// TwinCAT 3 PLC project Untitled1
// ProgramVersion: 3.1.4024.0
// libraries:
//   Tc2_Standard, * (Beckhoff Automation GmbH)
//   Tc2_System, * (Beckhoff Automation GmbH)
//   Tc3_Module, * (Beckhoff Automation GmbH)
// project tree:
//   GVLs/ GVL.TcGVL
//   / PlcTask.TcTTO
//   POUs/ MAIN.TcPOU, PLC_FB.TcPOU
// real-time tasks:
//   TASK PlcTask: cycle T#1ms, priority 20, ADS port 350
// I/O:
//   DEVICE Device 1 (EtherCAT), AmsNetId 5.136.192.215.2.1
//     Term 1 (EK1200) [EK1200-5000 EtherCAT Power supply (2A E-Bus)]
//       Term 2 (EL3104) [EL3104 4Ch. Ana. Input +/-10V Diff.]
//       Term 3 (EL1018) [EL1018 8Ch. Dig. Input 24V, 10µs]
//       Term 4 (EL2008) [EL2008 8Ch. Dig. Output 24V, 0.5A]
//       Term 5 (EL2008) [EL2008 8Ch. Dig. Output 24V, 0.5A]
//       Term 6 (EL2008) [EL2008 8Ch. Dig. Output 24V, 0.5A]
//       Term 7 (EL3632) [EL3632 2Ch. IEPE Sensor]
//       Term 8 (EL3632) [EL3632 2Ch. IEPE Sensor]
//       Term 9 (EL9011) [EL9011 End Terminal]
//   DEVICE Device 4 (COM Port)
//   DEVICE Device 5 (NOV-DP-RAM)
// variable links:
//   Untitled1/Untitled1 Instance <-> Device 1 (EtherCAT)/Term 1 (EK1200)/Term 2 (EL3104)
//     PlcTask Inputs/GVL.GvlDataAll[31] <-> AI Standard Channel 1/Value
//     PlcTask Inputs/GVL.GvlDataAll[32] <-> AI Standard Channel 2/Value
//     PlcTask Inputs/GVL.GvlDataAll[33] <-> AI Standard Channel 3/Value
//   Untitled1/Untitled1 Instance <-> Device 1 (EtherCAT)/Term 1 (EK1200)/Term 3 (EL1018)
//     PlcTask Inputs/GVL.Gvl_EL1018_FeedRead_Gray <-> Channel 1/Input
//     PlcTask Inputs/GVL.Gvl_EL1018_FeedRead_Gray @bit {1..7} <-> Channel {2..8}/Input  (7 links)
//   Untitled1/Untitled1 Instance <-> Device 1 (EtherCAT)/Term 1 (EK1200)/Term 4 (EL2008)
//     PlcTask Outputs/GVL.Gvl_EL2008_FeedWrite_Gray <-> Channel 1/Output
//     PlcTask Outputs/GVL.Gvl_EL2008_FeedWrite_Gray @bit {1..7} <-> Channel {2..8}/Output  (7 links)
//   Untitled1/Untitled1 Instance <-> Device 1 (EtherCAT)/Term 1 (EK1200)/Term 5 (EL2008)
//     PlcTask Outputs/GVL.Gvl_EL2008_SpindleWrite_Gray <-> Channel 1/Output
//     PlcTask Outputs/GVL.Gvl_EL2008_SpindleWrite_Gray @bit {1..7} <-> Channel {2..8}/Output  (7 links)
//   Untitled1/Untitled1 Instance <-> Device 1 (EtherCAT)/Term 1 (EK1200)/Term 6 (EL2008)
//     PlcTask Outputs/GVL.Gvl_Override_Valid <-> Channel 1/Output
//   Untitled1/Untitled1 Instance <-> Device 1 (EtherCAT)/Term 1 (EK1200)/Term 7 (EL3632)
//     PlcTask Inputs/GVL.GvlDataAll[10] <-> Ch1 Sample 9/Ch1 Value
//     PlcTask Inputs/GVL.GvlDataAll[11] <-> Ch2 Sample 0/Ch2 Value
//     PlcTask Inputs/GVL.GvlDataAll[12] <-> Ch2 Sample 1/Ch2 Value
//     PlcTask Inputs/GVL.GvlDataAll[13] <-> Ch2 Sample 2/Ch2 Value
//     PlcTask Inputs/GVL.GvlDataAll[14] <-> Ch2 Sample 3/Ch2 Value
//     PlcTask Inputs/GVL.GvlDataAll[15] <-> Ch2 Sample 4/Ch2 Value
//     PlcTask Inputs/GVL.GvlDataAll[16] <-> Ch2 Sample 5/Ch2 Value
//     PlcTask Inputs/GVL.GvlDataAll[17] <-> Ch2 Sample 6/Ch2 Value
//     PlcTask Inputs/GVL.GvlDataAll[18] <-> Ch2 Sample 7/Ch2 Value
//     PlcTask Inputs/GVL.GvlDataAll[19] <-> Ch2 Sample 8/Ch2 Value
//     PlcTask Inputs/GVL.GvlDataAll[1] <-> Ch1 Sample 0/Ch1 Value
//     PlcTask Inputs/GVL.GvlDataAll[20] <-> Ch2 Sample 9/Ch2 Value
//     PlcTask Inputs/GVL.GvlDataAll[2] <-> Ch1 Sample 1/Ch1 Value
//     PlcTask Inputs/GVL.GvlDataAll[3] <-> Ch1 Sample 2/Ch1 Value
//     PlcTask Inputs/GVL.GvlDataAll[4] <-> Ch1 Sample 3/Ch1 Value
//     PlcTask Inputs/GVL.GvlDataAll[5] <-> Ch1 Sample 4/Ch1 Value
//     PlcTask Inputs/GVL.GvlDataAll[6] <-> Ch1 Sample 5/Ch1 Value
//     PlcTask Inputs/GVL.GvlDataAll[7] <-> Ch1 Sample 6/Ch1 Value
//     PlcTask Inputs/GVL.GvlDataAll[8] <-> Ch1 Sample 7/Ch1 Value
//     PlcTask Inputs/GVL.GvlDataAll[9] <-> Ch1 Sample 8/Ch1 Value
//   Untitled1/Untitled1 Instance <-> Device 1 (EtherCAT)/Term 1 (EK1200)/Term 8 (EL3632)
//     PlcTask Inputs/GVL.GvlDataAll[{21..30}] <-> Ch1 Sample {0..9}/Ch1 Value  (10 links)

CONFIGURATION Untitled1
    RESOURCE PLC ON TwinCAT3
        TASK PlcTask(INTERVAL := T#1ms, PRIORITY := 20);
        PROGRAM MAIN WITH PlcTask : MAIN;
    END_RESOURCE
END_CONFIGURATION

// ---- GVLs/GVL.TcGVL
{attribute 'qualified_only'}
VAR_GLOBAL
	//================ 模拟量采集缓存 (核心业务) ================
	//硬件绑定变量     包含：2×EL3632振动模块 + 1×EL3104电流模块 + 其他模拟量输入
	//预定义80个INT数组，其中2个3632最多占用22个，3104占用4个
	GvlDataAll   AT%I*: ARRAY[1..80] OF INT;

	//缓存区变量
	//把 80 路模拟量（每路 100 个采样点）全缓存下来，方便做平均、滤波、FFT、包络等后处理
	GvlBuffer    AT%MB0: ARRAY[1..8000] OF INT;         //80通道模拟量缓存
	//16000 字节之后放 80 个 INT，用来记录“每一路当前写到了第几个采样
	//相当于 80 个“指针”，告诉程序每一路下一次该往 GvlBuffer 的哪个位置写新数据
	GvlIndexBuffer AT%MB16000: ARRAY[1..80] OF INT;  //数据索引
	
	
	//================ 上位机交互信号 (使用明确命名) ================
    // 进给倍率 (0-150%)
    Gvl_Cmd_FeedRate_Set    AT%I* : WORD; 
    
    // 主轴倍率 (0-120%)
    Gvl_Cmd_Spindle_Set     AT%I* : WORD;
    
    // [输出] 反馈给上位机的状态 (Actual)
    // 当前实际进给倍率 (EL1018读取并解码后的值)
    Gvl_Act_FeedRate_Real   AT%Q* : WORD;
	
	// 上位机决定是否启用倍率接管
    // TRUE = PLC接管机床倍率; FALSE = 机床使用自身面板倍率
    Gvl_Cmd_Enable_Override AT%I* : BOOL;

    //================ 硬件 I/O 映射 (倍率控制) ================
    // [输入] EL1018 读取机床当前的进给倍率波段 (原始格雷码)
    Gvl_EL1018_FeedRead_Gray AT%IB210 : BYTE; 

    // [输出] EL2008_1 向机床写入进给倍率 (转换后的格雷码)
    Gvl_EL2008_FeedWrite_Gray AT%QB71 : BYTE;

    // [输出] EL2008_2 向机床写入主轴倍率 (转换后的格雷码)
    Gvl_EL2008_SpindleWrite_Gray AT%QB72 : BYTE;

    // [输出] 倍率有效信号
    Gvl_Override_Valid AT%QX73.0 : BOOL;
	
END_VAR

// ---- POUs/MAIN.TcPOU
PROGRAM MAIN
VAR
	plc_fb:PLC_FB;
END_VAR

plc_fb
(
	//功能块输入参数
	PlcDataAll:=GVL.GvlDataAll,
    //功能块输出参数
	PlcBuffer=>Gvl.GvlBuffer,
	IndexBuffer=>Gvl.GvlIndexBuffer,
	
	// === 交互部分 ===
    Cmd_FeedRate     := GVL.Gvl_Cmd_FeedRate_Set,
    Cmd_SpindleSpeed := GVL.Gvl_Cmd_Spindle_Set,
    
    // 【新增】绑定上位机使能信号
    Cmd_Enable       := GVL.Gvl_Cmd_Enable_Override, 
    
    Act_FeedRate     => GVL.Gvl_Act_FeedRate_Real,
    
    // === 硬件IO部分 ===
    RawFeedRead_Gray     := GVL.Gvl_EL1018_FeedRead_Gray,
    OutFeedWrite_Gray    => GVL.Gvl_EL2008_FeedWrite_Gray,
    OutSpindleWrite_Gray => GVL.Gvl_EL2008_SpindleWrite_Gray,
    
    // 【修改】硬件有效位现在由 FB 的逻辑决定
    OutOverrideValid     => GVL.Gvl_Override_Valid

);

END_PROGRAM

// ---- POUs/PLC_FB.TcPOU
FUNCTION_BLOCK PLC_FB
VAR_INPUT
	PlcDataAll: ARRAY[1..80] OF INT;    //80模拟量采集通道	
	// === 上位机指令 ===
    Cmd_FeedRate     : WORD;  //设定进给倍率
    Cmd_SpindleSpeed : WORD;  //设定主轴转速倍率
    Cmd_Enable       : BOOL;  // 接收上位机的使能信号
	
	// === 硬件原始输入 ===
    RawFeedRead_Gray : BYTE;
END_VAR

VAR_OUTPUT
	PlcBuffer: ARRAY[1..8000] OF INT;    // 80×100 环形缓存
	IndexBuffer: ARRAY[1..80] OF INT;    // 每路内部的 1-based 写指针（1~100）
	
	Act_FeedRate     : WORD;  
    // === 硬件输出 ===
    OutFeedWrite_Gray    : BYTE;
    OutSpindleWrite_Gray : BYTE;
    OutOverrideValid     : BOOL; 
END_VAR

VAR
    {* 循环/计算用局部变量 *}
    i      : INT;      // 循环计数（1..80）
	
    tempBin  : BYTE;
    TargetFeedBin    : WORD;
    TargetSpindleBin : WORD;
END_VAR

//***********模拟量存入缓存区 BEGIN***********//
{* ============  80 路环形缓存  ============ *}
FOR i := 1 TO 80 DO
    // 确保指针有效
    IF IndexBuffer[i] < 1 THEN
        IndexBuffer[i] := 1;
    ELSIF IndexBuffer[i] > 100 THEN
        IndexBuffer[i] := 1;
    END_IF;

    // 写入：本路基地址 + 偏移
    PlcBuffer[(i - 1) * 100 + IndexBuffer[i]] := PlcDataAll[i];

    // 更新指针
    IndexBuffer[i] := IndexBuffer[i] + 1;
    IF IndexBuffer[i] > 100 THEN
        IndexBuffer[i] := 1;
    END_IF;
END_FOR;
{* ============  环形缓存结束  ============ *}
//***********模拟量存入缓存区 END***********//


//=========================================================
// 2. 倍率读取逻辑 (EL1018 -> 取反解码 -> 上位机)
//=========================================================
// 【修改点】既然验证了 0%=255, 200%=55，说明是二进制取反逻辑
// 使用 NOT 指令直接还原真实值
tempBin := NOT RawFeedRead_Gray;

// B. 根据是否使能，决定反馈给上位机显示什么值
IF Cmd_Enable THEN
    // 情况1：PLC接管时，反馈“设定值”，保证界面显示稳定
    Act_FeedRate := Cmd_FeedRate;
ELSE
    // 情况2：面板控制时，反馈“硬件读取值”
    Act_FeedRate := BYTE_TO_WORD(tempBin);
END_IF;

// 【注意】原代码这里有一句重复赋值导致逻辑覆盖，已删除


//=========================================================
// 3. 倍率写入逻辑 (PLC -> 取反编码 -> EL2008)
//=========================================================
TargetFeedBin    := Cmd_FeedRate;
TargetSpindleBin := Cmd_SpindleSpeed;

// -- 进给倍率写入 --
// 限制最大值防止溢出 (根据你测得的 200% = 200，这里最大可以放宽，但Byte上限是255)
IF TargetFeedBin > 255 THEN TargetFeedBin := 255; END_IF;

// 【修改点】既然输入是反码，输出给机床也必须是反码
// 例如：设定 100 (01100100) -> 发送 NOT -> 155 (10011011)
OutFeedWrite_Gray := NOT WORD_TO_BYTE(TargetFeedBin);


// -- 主轴倍率写入 --
// 【注意】假设主轴倍率开关原理和进给一样，也改为取反逻辑
// 如果主轴读数不对，请改回原来的格雷码逻辑
IF TargetSpindleBin > 255 THEN TargetSpindleBin := 255; END_IF;
OutSpindleWrite_Gray := NOT WORD_TO_BYTE(TargetSpindleBin);


//=========================================================
// 4. 有效位控制逻辑
//=========================================================
// 只有当上位机置位 Cmd_Enable 为 TRUE 时，硬件输出才生效
OutOverrideValid := Cmd_Enable;

END_FUNCTION_BLOCK
